LIN {X 0,Y 90.915,Z 523.558,A -85,B 0,C 180,E1 -30409.92,E2 -30409.92} C_VEL
LIN {X 0,Y 93.111,Z 505.621,A -85,B 0,C 180,E1 -30410.51,E2 -30410.51} C_VEL
LIN {X 0,Y 91.871,Z 501.281,A -85,B 0,C 180,E1 -30415.076,E2 -30415.076} C_VEL
LIN {X 0,Y 91.126,Z 498.615,A -85,B 0,C 180,E1 -30419.189,E2 -30419.189} C_VEL
LIN {X 0,Y 90.737,Z 496.287,A -85,B 0,C 180,E1 -30424.442,E2 -30424.442} C_VEL
LIN {X 0,Y 90.686,Z 496.641,A -85,B 0,C 180,E1 -30428.635,E2 -30428.635} C_VEL
LIN {X 0,Y 91.413,Z 499.975,A -85,B 0,C 180,E1 -30436.039,E2 -30436.039} C_VEL
LIN {X 0,Y 92.407,Z 503.34,A -85,B 0,C 180,E1 -30440.415,E2 -30440.415} C_VEL
LIN {X 0,Y 93.073,Z 505.914,A -85,B 0,C 180,E1 -30442.748,E2 -30442.748} C_VEL
LIN {X 0,Y 90.759,Z 523.808,A -85,B 0,C 180,E1 -30443.218,E2 -30443.218} C_VEL
LIN {X 0,Y 87.684,Z 537.514,A -85,B 0,C 180,E1 -30443.97,E2 -30443.97} C_VEL
LIN {X 0,Y 83.772,Z 549.3,A -85,B 0,C 180,E1 -30444.902,E2 -30444.902} C_VEL
LIN {X 0,Y 78.485,Z 561.315,A -85,B 0,C 180,E1 -30446.432,E2 -30446.432} C_VEL
LIN {X 0,Y 71.934,Z 572.842,A -85,B 0,C 180,E1 -30448.44,E2 -30448.44} C_VEL
LIN {X 0,Y 66.282,Z 581.074,A -85,B 0,C 180,E1 -30450.512,E2 -30450.512} C_VEL
LIN {X 0,Y 63.358,Z 584.941,A -85,B 0,C 180,E1 -30451.848,E2 -30451.848} C_VEL
LIN {X 0,Y 59.505,Z 589.3,A -85,B 0,C 180,E1 -30453.039,E2 -30453.039} C_VEL
LIN {X 0,Y 52.127,Z 595.921,A -85,B 0,C 180,E1 -30453.76,E2 -30453.76} C_VEL
LIN {X 0,Y 44.318,Z 601.959,A -85,B 0,C 180,E1 -30454.921,E2 -30454.921} C_VEL
LIN {X 0,Y 39.873,Z 605.38,A -85,B 0,C 180,E1 -30457.338,E2 -30457.338} C_VEL
LIN {X 0,Y 31.277,Z 611.937,A -85,B 0,C 180,E1 -30467.613,E2 -30467.613} C_VEL
LIN {X 0,Y 24.232,Z 617.099,A -85,B 0,C 180,E1 -30484.208,E2 -30484.208} C_VEL
LIN {X 0,Y 20.914,Z 619.883,A -85,B 0,C 180,E1 -30500.313,E2 -30500.313} C_VEL
LIN {X 0,Y 19.526,Z 623.216,A -85,B 0,C 180,E1 -30531.089,E2 -30531.089} C_VEL
LIN {X 0,Y 21.628,Z 624.874,A -85,B 0,C 180,E1 -30550.526,E2 -30550.526} C_VEL
LIN {X 0,Y 26.715,Z 626.316,A -85,B 0,C 180,E1 -30568.256,E2 -30568.256} C_VEL
LIN {X 0,Y 36.599,Z 627.259,A -85,B 0,C 180,E1 -30583.752,E2 -30583.752} C_VEL
LIN {X 0,Y 46.075,Z 627.038,A -85,B 0,C 180,E1 -30591.227,E2 -30591.227} C_VEL
LIN {X 0,Y 56.342,Z 625.845,A -85,B 0,C 180,E1 -30596.25,E2 -30596.25} C_VEL
LIN {X 0,Y 68.01,Z 623.359,A -85,B 0,C 180,E1 -30600.001,E2 -30600.001} C_VEL
LIN {X 0,Y 80.919,Z 619.2,A -85,B 0,C 180,E1 -30602.86,E2 -30602.86} C_VEL
LIN {X 0,Y 91.649,Z 614.469,A -85,B 0,C 180,E1 -30604.549,E2 -30604.549} C_VEL
LIN {X 0,Y 102.959,Z 608.086,A -85,B 0,C 180,E1 -30605.942,E2 -30605.942} C_VEL
LIN {X 0,Y 101.089,Z 609.294,A -85,B 0,C 180,E1 -30606.709,E2 -30606.709} C_VEL
LIN {X 0,Y 92.189,Z 614.244,A -85,B 0,C 180,E1 -30607.688,E2 -30607.688} C_VEL
LIN {X 0,Y 81.883,Z 618.911,A -85,B 0,C 180,E1 -30609.249,E2 -30609.249} C_VEL
LIN {X 0,Y 71.677,Z 622.492,A -85,B 0,C 180,E1 -30611.342,E2 -30611.342} C_VEL
LIN {X 0,Y 64.94,Z 624.354,A -85,B 0,C 180,E1 -30613.106,E2 -30613.106} C_VEL
LIN {X 0,Y 51.682,Z 626.784,A -85,B 0,C 180,E1 -30617.855,E2 -30617.855} C_VEL
LIN {X 0,Y 39.058,Z 627.687,A -85,B 0,C 180,E1 -30625.891,E2 -30625.891} C_VEL
LIN {X 0,Y 33.24,Z 627.55,A -85,B 0,C 180,E1 -30632.257,E2 -30632.257} C_VEL
LIN {X 0,Y 23.729,Z 626.099,A -85,B 0,C 180,E1 -30653.681,E2 -30653.681} C_VEL
LIN {X 0,Y 20.902,Z 624.797,A -85,B 0,C 180,E1 -30670.358,E2 -30670.358} C_VEL
LIN {X 0,Y 19.978,Z 623.07,A -85,B 0,C 180,E1 -30690.005,E2 -30690.005} C_VEL
LIN {X 0,Y 21.941,Z 619.571,A -85,B 0,C 180,E1 -30718.721,E2 -30718.721} C_VEL
LIN {X 0,Y 27.789,Z 614.941,A -85,B 0,C 180,E1 -30739.355,E2 -30739.355} C_VEL
LIN {X 0,Y 37.312,Z 607.914,A -85,B 0,C 180,E1 -30753.473,E2 -30753.473} C_VEL
LIN {X 0,Y 46.518,Z 600.286,A -85,B 0,C 180,E1 -30760.781,E2 -30760.781} C_VEL
LIN {X 0,Y 54.243,Z 592.719,A -85,B 0,C 180,E1 -30765.099,E2 -30765.099} C_VEL
LIN {X 0,Y 62.794,Z 582.855,A -85,B 0,C 180,E1 -30768.328,E2 -30768.328} C_VEL
LIN {X 0,Y 69.493,Z 573.477,A -85,B 0,C 180,E1 -30770.419,E2 -30770.419} C_VEL
LIN {X 0,Y 76.319,Z 561.926,A -85,B 0,C 180,E1 -30771.865,E2 -30771.865} C_VEL
LIN {X 0,Y 81.871,Z 549.729,A -85,B 0,C 180,E1 -30773.006,E2 -30773.006} C_VEL
LIN {X 0,Y 86.267,Z 536.474,A -85,B 0,C 180,E1 -30773.824,E2 -30773.824} C_VEL
LIN {X 0,Y 89.219,Z 523.153,A -85,B 0,C 180,E1 -30774.3,E2 -30774.3} C_VEL
LIN {X 0,Y 90.931,Z 509.494,A -85,B 0,C 180,E1 -30774.762,E2 -30774.762} C_VEL
LIN {X 0,Y 90.128,Z 505.651,A -85,B 0,C 180,E1 -30779.795,E2 -30779.795} C_VEL
LIN {X 0,Y 89.838,Z 503.497,A -85,B 0,C 180,E1 -30784.486,E2 -30784.486} C_VEL
LIN {X 0,Y 89.787,Z 503.623,A -85,B 0,C 180,E1 -30787.873,E2 -30787.873} C_VEL
LIN {X 0,Y 90.248,Z 506.626,A -85,B 0,C 180,E1 -30794.66,E2 -30794.66} C_VEL
LIN {X 0,Y 90.913,Z 509.501,A -85,B 0,C 180,E1 -30798.439,E2 -30798.439} C_VEL
LIN {X 0,Y 89.595,Z 520.258,A -85,B 0,C 180,E1 -30798.795,E2 -30798.795} C_VEL
LIN {X 0,Y 86.93,Z 533.67,A -85,B 0,C 180,E1 -30799.232,E2 -30799.232} C_VEL
LIN {X 0,Y 83.208,Z 545.699,A -85,B 0,C 180,E1 -30799.874,E2 -30799.874} C_VEL
LIN {X 0,Y 78.119,Z 557.906,A -85,B 0,C 180,E1 -30801.024,E2 -30801.024} C_VEL
LIN {X 0,Y 72.235,Z 568.844,A -85,B 0,C 180,E1 -30802.438,E2 -30802.438} C_VEL
LIN {X 0,Y 65.433,Z 578.946,A -85,B 0,C 180,E1 -30804.08,E2 -30804.08} C_VEL
LIN {X 0,Y 58.869,Z 587.203,A -85,B 0,C 180,E1 -30806.442,E2 -30806.442} C_VEL
LIN {X 0,Y 50.734,Z 595.826,A -85,B 0,C 180,E1 -30810.026,E2 -30810.026} C_VEL
LIN {X 0,Y 41.337,Z 604.19,A -85,B 0,C 180,E1 -30816.138,E2 -30816.138} C_VEL
LIN {X 0,Y 39.873,Z 605.38,A -85,B 0,C 180,E1 -30817.338,E2 -30817.338} C_VEL
LIN {X 0,Y 35.421,Z 608.646,A -85,B 0,C 180,E1 -30820.552,E2 -30820.552} C_VEL
LIN {X 0,Y 27.181,Z 613.412,A -85,B 0,C 180,E1 -30825.598,E2 -30825.598} C_VEL
LIN {X 0,Y 20.452,Z 616.689,A -85,B 0,C 180,E1 -30832.342,E2 -30832.342} C_VEL
LIN {X 0,Y 14.847,Z 619.562,A -85,B 0,C 180,E1 -30848.292,E2 -30848.292} C_VEL
LIN {X 0,Y 12.281,Z 622.59,A -85,B 0,C 180,E1 -30886.617,E2 -30886.617} C_VEL
LIN {X 0,Y 16.748,Z 625.154,A -85,B 0,C 180,E1 -30927.049,E2 -30927.049} C_VEL
LIN {X 0,Y 22.559,Z 626.365,A -85,B 0,C 180,E1 -30941.85,E2 -30941.85} C_VEL
LIN {X 0,Y 35.251,Z 627.383,A -85,B 0,C 180,E1 -30955.398,E2 -30955.398} C_VEL
LIN {X 0,Y 44.257,Z 627.171,A -85,B 0,C 180,E1 -30960.001,E2 -30960.001} C_VEL
LIN {X 0,Y 56.346,Z 625.811,A -85,B 0,C 180,E1 -30963.813,E2 -30963.813} C_VEL
LIN {X 0,Y 67.173,Z 623.558,A -85,B 0,C 180,E1 -30966.006,E2 -30966.006} C_VEL
LIN {X 0,Y 63.706,Z 624.43,A -85,B 0,C 180,E1 -30966.87,E2 -30966.87} C_VEL
LIN {X 0,Y 49.961,Z 626.773,A -85,B 0,C 180,E1 -30970.056,E2 -30970.056} C_VEL
LIN {X 0,Y 36.519,Z 627.593,A -85,B 0,C 180,E1 -30975.808,E2 -30975.808} C_VEL
LIN {X 0,Y 23.946,Z 626.823,A -85,B 0,C 180,E1 -30988.311,E2 -30988.311} C_VEL
LIN {X 0,Y 14.427,Z 624.533,A -85,B 0,C 180,E1 -31020.855,E2 -31020.855} C_VEL
LIN {X 0,Y 12.897,Z 622.731,A -85,B 0,C 180,E1 -31050.008,E2 -31050.008} C_VEL
LIN {X 0,Y 16.065,Z 619.153,A -85,B 0,C 180,E1 -31091.019,E2 -31091.019} C_VEL
LIN {X 0,Y 23.756,Z 614.431,A -85,B 0,C 180,E1 -31112.571,E2 -31112.571} C_VEL
LIN {X 0,Y 34.712,Z 607.308,A -85,B 0,C 180,E1 -31124.103,E2 -31124.103} C_VEL
LIN {X 0,Y 44.681,Z 599.549,A -85,B 0,C 180,E1 -31129.448,E2 -31129.448} C_VEL
LIN {X 0,Y 50.908,Z 593.751,A -85,B 0,C 180,E1 -31132.064,E2 -31132.064} C_VEL
LIN {X 0,Y 58.302,Z 585.942,A -85,B 0,C 180,E1 -31133.987,E2 -31133.987} C_VEL
LIN {X 0,Y 66.059,Z 576.028,A -85,B 0,C 180,E1 -31135.873,E2 -31135.873} C_VEL
LIN {X 0,Y 73.025,Z 565.187,A -85,B 0,C 180,E1 -31136.865,E2 -31136.865} C_VEL
LIN {X 0,Y 78.231,Z 555.01,A -85,B 0,C 180,E1 -31137.59,E2 -31137.59} C_VEL
LIN {X 0,Y 82.798,Z 543.518,A -85,B 0,C 180,E1 -31138.175,E2 -31138.175} C_VEL
LIN {X 0,Y 86.215,Z 531.759,A -85,B 0,C 180,E1 -31138.592,E2 -31138.592} C_VEL
LIN {X 0,Y 88.722,Z 518.174,A -85,B 0,C 180,E1 -31138.909,E2 -31138.909} C_VEL
LIN {X 0,Y 89.235,Z 513.755,A -85,B 0,C 180,E1 -31139.16,E2 -31139.16} C_VEL
LIN {X 0,Y 88.969,Z 511.732,A -85,B 0,C 180,E1 -31142.546,E2 -31142.546} C_VEL
LIN {X 0,Y 88.923,Z 510.489,A -85,B 0,C 180,E1 -31145.669,E2 -31145.669} C_VEL
LIN {X 0,Y 88.89,Z 510.742,A -85,B 0,C 180,E1 -31147.381,E2 -31147.381} C_VEL
LIN {X 0,Y 89.134,Z 513.296,A -85,B 0,C 180,E1 -31153.247,E2 -31153.247} C_VEL
LIN {X 0,Y 89.226,Z 513.943,A -85,B 0,C 180,E1 -31154.167,E2 -31154.167} C_VEL
LIN {X 0,Y 87.085,Z 527.705,A -85,B 0,C 180,E1 -31154.435,E2 -31154.435} C_VEL
LIN {X 0,Y 83.902,Z 539.922,A -85,B 0,C 180,E1 -31154.824,E2 -31154.824} C_VEL
LIN {X 0,Y 80.16,Z 550.289,A -85,B 0,C 180,E1 -31155.33,E2 -31155.33} C_VEL
LIN {X 0,Y 74.145,Z 562.9,A -85,B 0,C 180,E1 -31156.313,E2 -31156.313} C_VEL
LIN {X 0,Y 67.216,Z 574.178,A -85,B 0,C 180,E1 -31157.427,E2 -31157.427} C_VEL
LIN {X 0,Y 62.036,Z 581.141,A -85,B 0,C 180,E1 -31158.413,E2 -31158.413} C_VEL
LIN {X 0,Y 54.34,Z 589.997,A -85,B 0,C 180,E1 -31160.333,E2 -31160.333} C_VEL
LIN {X 0,Y 45.911,Z 598.122,A -85,B 0,C 180,E1 -31163.294,E2 -31163.294} C_VEL
LIN {X 0,Y 35.929,Z 606.112,A -85,B 0,C 180,E1 -31168.326,E2 -31168.326} C_VEL
LIN {X 0,Y 26.437,Z 612.476,A -85,B 0,C 180,E1 -31177.1,E2 -31177.1} C_VEL
LIN {X 0,Y 18.039,Z 617.541,A -85,B 0,C 180,E1 -31194.233,E2 -31194.233} C_VEL
LIN {X 0,Y 14.847,Z 619.562,A -85,B 0,C 180,E1 -31208.292,E2 -31208.292} C_VEL
LIN {X 0,Y 11.93,Z 621.465,A -85,B 0,C 180,E1 -31228.973,E2 -31228.973} C_VEL
LIN {X 0,Y 10.643,Z 624.035,A -85,B 0,C 180,E1 -31278.768,E2 -31278.768} C_VEL
LIN {X 0,Y 14.859,Z 625.567,A -85,B 0,C 180,E1 -31309.233,E2 -31309.233} C_VEL
LIN {X 0,Y 19.891,Z 626.386,A -85,B 0,C 180,E1 -31319.482,E2 -31319.482} C_VEL
LIN {X 0,Y 21.758,Z 626.591,A -85,B 0,C 180,E1 -31321.236,E2 -31321.236} C_VEL
LIN {X 0,Y 28.214,Z 627.217,A -85,B 0,C 180,E1 -31324.923,E2 -31324.923} C_VEL
LIN {X 0,Y 28.324,Z 627.24,A -85,B 0,C 180,E1 -31327.06,E2 -31327.06} C_VEL
LIN {X 0,Y 14.889,Z 625.645,A -85,B 0,C 180,E1 -31339.281,E2 -31339.281} C_VEL
LIN {X 0,Y 8.919,Z 624.246,A -85,B 0,C 180,E1 -31358.024,E2 -31358.024} C_VEL
LIN {X 0,Y 5.802,Z 622.392,A -85,B 0,C 180,E1 -31410.017,E2 -31410.017} C_VEL
LIN {X 0,Y 11.673,Z 618.732,A -85,B 0,C 180,E1 -31474.583,E2 -31474.583} C_VEL
LIN {X 0,Y 21.423,Z 613.92,A -85,B 0,C 180,E1 -31489.813,E2 -31489.813} C_VEL
LIN {X 0,Y 31.734,Z 607.833,A -85,B 0,C 180,E1 -31495.293,E2 -31495.293} C_VEL
LIN {X 0,Y 42.187,Z 600.229,A -85,B 0,C 180,E1 -31498.307,E2 -31498.307} C_VEL
LIN {X 0,Y 50.777,Z 592.584,A -85,B 0,C 180,E1 -31500.155,E2 -31500.155} C_VEL
LIN {X 0,Y 58.872,Z 583.957,A -85,B 0,C 180,E1 -31501.172,E2 -31501.172} C_VEL
LIN {X 0,Y 66.813,Z 573.552,A -85,B 0,C 180,E1 -31502.135,E2 -31502.135} C_VEL
LIN {X 0,Y 73.866,Z 562.061,A -85,B 0,C 180,E1 -31502.533,E2 -31502.533} C_VEL
LIN {X 0,Y 79.455,Z 550.375,A -85,B 0,C 180,E1 -31502.937,E2 -31502.937} C_VEL
LIN {X 0,Y 83.893,Z 537.789,A -85,B 0,C 180,E1 -31503.245,E2 -31503.245} C_VEL
LIN {X 0,Y 87.125,Z 524.219,A -85,B 0,C 180,E1 -31503.41,E2 -31503.41} C_VEL
LIN {X 0,Y 88.001,Z 518.595,A -85,B 0,C 180,E1 -31503.537,E2 -31503.537} C_VEL
LIN {X 0,Y 88.033,Z 517.628,A -85,B 0,C 180,E1 -31505.727,E2 -31505.727} C_VEL
LIN {X 0,Y 87.934,Z 518.676,A -85,B 0,C 180,E1 -31508.908,E2 -31508.908} C_VEL
LIN {X 0,Y 87.938,Z 518.969,A -85,B 0,C 180,E1 -31509.636,E2 -31509.636} C_VEL
LIN {X 0,Y 85.276,Z 532.679,A -85,B 0,C 180,E1 -31509.843,E2 -31509.843} C_VEL
LIN {X 0,Y 81.521,Z 544.947,A -85,B 0,C 180,E1 -31510.053,E2 -31510.053} C_VEL
LIN {X 0,Y 75.972,Z 557.885,A -85,B 0,C 180,E1 -31510.598,E2 -31510.598} C_VEL
LIN {X 0,Y 69.843,Z 568.867,A -85,B 0,C 180,E1 -31511.158,E2 -31511.158} C_VEL
LIN {X 0,Y 62.78,Z 579.003,A -85,B 0,C 180,E1 -31511.609,E2 -31511.609} C_VEL
LIN {X 0,Y 55.806,Z 587.283,A -85,B 0,C 180,E1 -31512.575,E2 -31512.575} C_VEL
LIN {X 0,Y 47.065,Z 595.932,A -85,B 0,C 180,E1 -31513.918,E2 -31513.918} C_VEL
LIN {X 0,Y 36.614,Z 604.317,A -85,B 0,C 180,E1 -31516.309,E2 -31516.309} C_VEL
LIN {X 0,Y 26.276,Z 611.064,A -85,B 0,C 180,E1 -31520.581,E2 -31520.581} C_VEL
LIN {X 0,Y 16.173,Z 616.455,A -85,B 0,C 180,E1 -31529.635,E2 -31529.635} C_VEL
LIN {X 0,Y 9.832,Z 619.411,A -85,B 0,C 180,E1 -31544.361,E2 -31544.361} C_VEL
LIN {X 0,Y 5.696,Z 622.932,A -85,B 0,C 180,E1 -31628.071,E2 -31628.071} C_VEL
LIN {X 0,Y 14.161,Z 625.427,A -85,B 0,C 180,E1 -31672.936,E2 -31672.936} C_VEL
LIN {X 0,Y 21.758,Z 626.591,A -85,B 0,C 180,E1 -31681.236,E2 -31681.236} C_VEL
LIN {X 0,Y 21.758,Z 626.591,A -85,B 0,C 180,E1 -31681.236,E2 -31681.236}

QRS_NEXT_CUT()

QRS_NEXT()
QRS_HOME()

END
